{attribute addProperty BoxType "EL6201-0000-0017"}
{attribute addProperty Id "Slave_12A_DI0BIT10.12589Slave_12A_DI1BIT10.12590Slave_12A_DI2BIT10.12591Slave_12A_DI3BIT10.12592Slave_12B_DI0BIT10.12593Slave_12B_DI1BIT10.12594Slave_12B_DI2BIT10.12595Slave_12B_DI3BIT10.12596"}
{attribute addProperty CRC "335435865"}
{attribute addProperty SizeInBites "8"}
{attribute addProperty SizeInBytes "1"}
TYPE Slave_12_Inputs_13FE5859 :
STRUCT
	{attribute addProperty Name "Slave_12A_DI0"}
	Slave_12A_DI0 : BIT;
	{attribute addProperty Name "Slave_12A_DI1"}
	Slave_12A_DI1 : BIT;
	{attribute addProperty Name "Slave_12A_DI2"}
	Slave_12A_DI2 : BIT;
	{attribute addProperty Name "Slave_12A_DI3"}
	Slave_12A_DI3 : BIT;
	{attribute addProperty Name "Slave_12B_DI0"}
	Slave_12B_DI0 : BIT;
	{attribute addProperty Name "Slave_12B_DI1"}
	Slave_12B_DI1 : BIT;
	{attribute addProperty Name "Slave_12B_DI2"}
	Slave_12B_DI2 : BIT;
	{attribute addProperty Name "Slave_12B_DI3"}
	Slave_12B_DI3 : BIT;
END_STRUCT
END_TYPE

(* stored: Version 1.2.0.0, ProductVersion 3.1.4024.9
   DUT Slave_12_Inputs_13FE5859: Id {8675fb0b-3648-4e2a-b656-383f34c4b750} *)
